TYPE ST_SerLVC4000 :
STRUCT
    (* Readbacks *)
    {attribute 'pytmc' := '
    pv: voltage;
    io: i;
    '}
    i_iOut	:	INT; //Output voltage
    (* Controls *)
    {attribute 'pytmc' := '
    pv: ADC_COEFF;
    io: io;
    '}
    q_rADCsl	:	REAL; //ADC slope coeff
    {attribute 'pytmc' := '
    pv: ADC_OFFSET;
    io: io;
    '}
    q_rADCos	:	REAL; //ADC offset
    {attribute 'pytmc' := '
    pv: CALIB_SET;
    io: io;
    '}
    q_xCal	:	BOOL; //Activate calibration mode
    {attribute 'pytmc' := '
    pv: DISP_SET;
    io: io;
    '}
    q_xFull	:	BOOL; //Set full displacement during calibration
    {attribute 'pytmc' := '
    pv: ZERO_SET;
    io: io;
    '}
    q_xZero	:	BOOL; //Set zero during calibration
    {attribute 'pytmc' := '
    pv: GAIN_SET;
    io: io;
    '}
    q_iGain	:	INT; //Set instrument gain
    {attribute 'pytmc' := '
    pv: CALIB_ABORT;
    io: io;
    '}
    q_xAbortCal	:	BOOL; //Abort calibration mode
    (* Internal params *)
    {attribute 'pytmc' := '
    pv: ADDR;
    io: io;
    '}
    iAddr	:	INT; //RS485 address
    xTimeout	:	BOOL; //Timeout (true if no comm)
END_STRUCT
END_TYPE

(* stored: Version 1.1.0.1, ProductVersion 3.1.4022.16
   DUT ST_SerLVC4000: Id {1ecc4b20-fded-4e3a-82c1-cf810d73e466} *)
